KUKA KRL program: LAB_MISSING_TARGET.src, LAB_MISSING_TARGET.dat

--- LAB_MISSING_TARGET.src ---
&ACCESS RVP
&REL 1
&PARAM TEMPLATE = C:\KRC\Roboter\Template\vorgabe
&PARAM EDITMASK = *
DEF LAB_MISSING_TARGET()
  ; KLAB fixture: intentional unresolved target
  BAS(#INITMOV,0)
  $ADVANCE=3
  $IPO_MODE=#BASE
  BAS(#TOOL,0)
  BAS(#BASE,0)
  BAS(#VEL_PTP,20)
  BAS(#ACC_PTP,20)
  $VEL.CP=0.1
  LIN P_MISSING
END

--- LAB_MISSING_TARGET.dat ---
&ACCESS RVP
&REL 1
DEFDAT LAB_MISSING_TARGET PUBLIC
  DECL E6AXIS A_HOME={A1 0,A2 -90,A3 90,A4 0,A5 0,A6 0,E1 0,E2 0,E3 0,E4 0,E5 0,E6 0}
ENDDAT
